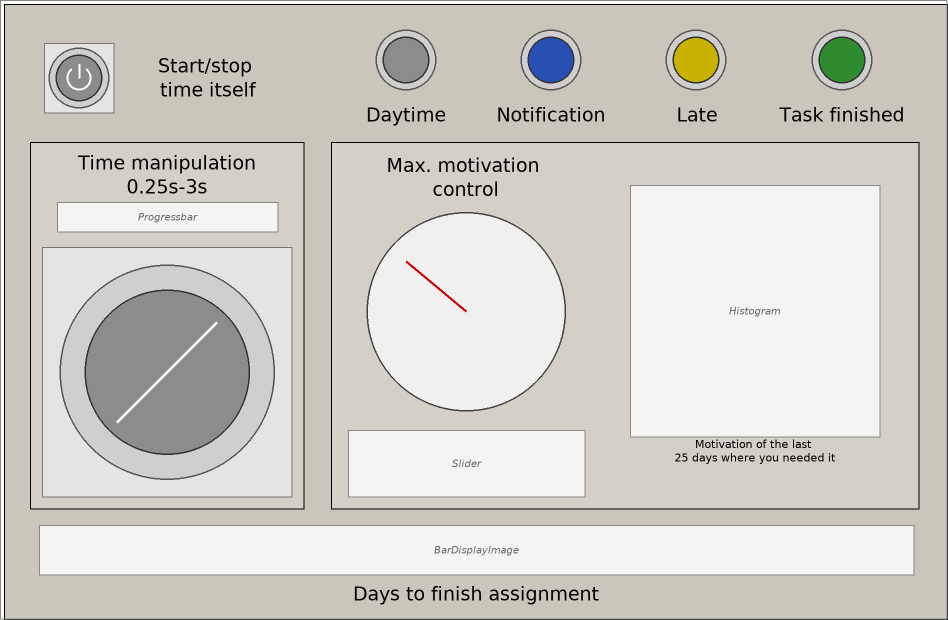
VISUALIZATION Visualization  // 948x620
    Rectangle (4,4 944x616)
    RoundedRectangle (331,142 588x367)
    RoundedRectangle (30,142 274x367)
    Label (133,51 150x54), "Start/stop time itself"
    PowerSwitch (44,43 70x70), variable: Calender.On, behaviour: TOGGLE, style: Switch-PowerSwitch-Gray
    Progressbar (57,202 221x30), variable: Calender.HalfADay
    Label (70,153 194x44), "Time manipulation 0.25s-3s"
    Potentiometer360 (42,247 250x250), variable: Calender.HalfADay, style: Potentiometer-Potentiometer360-Gray, scale format: %.1f, scale 250..2250
        p518627256: [ms]
    Histogram (630,185 250x252), scale format: %.1f, scale 0..100
        p1518820177: Student.MotivationTracker
        p102497268: Student.MotivationTracker
        p788070771: ARRAY [1..25] OF INT
    Label (674,436 162x30), "Motivation of the last 25 days where you needed it"
    Meter360 (363,212 206x199), value: Student.Motivation, style: Meter-Meter360-Gray, scale format: %.1f, scale 0..100
        p518627256: Motivation amount
    Slider (348,430 237x67), variable: Student.MaxMotivation1, scale 0..100
    Label (336,152 260x51), "Max. motivation control"
    Label (331,100 150x30), "Daytime"
    Label (767,100 150x30), "Task finished"
    Label (622,100 150x30), "Late"
    Label (476,100 150x30), "Notification"
    Lamp1 (371,25 70x70), variable: Calender.calenderTimer.IN, style: Lamp-Lamp1-Gray
    Lamp1 (807,25 70x70), variable: GVL.Finished, style: Lamp-Lamp1-Green
    Lamp1 (661,25 70x70), variable: brightspace.Late, style: Lamp-Lamp1-Yellow
    Lamp1 (516,25 70x70), variable: Student.StudentNotification, style: Lamp-Lamp1-Blue
    BarDisplayImage (39,525 875x50), value: GVL.MainDueIn, style: BarDisplayImage-Gray, scale format: %.1f, scale -30..30
    Label (328,579 296x30), "Days to finish assignment"
END_VISUALIZATION

(* stored: Version 1.1.0.1, ProductVersion 3.1.4024.12
   Visu Visualization: Id {e2cdd09a-e53f-46bc-af50-254e2307d941} *)
